TYPE
  ST_FaultRecord : STRUCT
  nFaultCode : UINT; // 故障代码
  tFaultTime : TIME; // 故障发生时间
  eFaultType : E_FaultType; // 故障类型
  bActive : BOOL; // 是否为当前活跃故障
  sDescription : STRING(80); // 故障描述
END_STRUCT;
END_TYPE

(* stored: Version 1.1.0.1, ProductVersion 3.1.4024.12
   DUT ST_FaultRecord: Id {550e8400-e29b-41d4-a716-446655440003}, Type STRUCT *)
